// Mitsubishi GX Works2 project: 051023 aula antes de apagar   PLC: Q03UDV

// task Task_01 (event TRUE, interval 0, priority 31): 
// task ST_Example_Safe (event TRUE, interval 0, priority 31): ST_Example_Safe

PROGRAM ST_Example_Safe
VAR
  iDR : INT;
  iHabilitar : BOOL;
  stgOperador : STRING[32];
  iValor01 : INT;
  iValor02 : INT;
END_VAR
iDR:= fEscolherOperacao1( iHabilitar , stgOperador , iValor01 , iValor02 );

iDR:= fEscolherOperacao2( iHabilitar , stgOperador , iValor01 , iValor02 );
END_PROGRAM

FUNCTION fEscolherOperacao1
VAR_INPUT
  xHabilitar : BOOL;
  stgoperador : STRING[32];
  iValor01 : INT;
  iValor02 : INT;
END_VAR
IF xHabilitar THEN 	
	IF  stgoperador="+"  THEN
			 fEscolherOperacao1:=iValor01+iValor02;
	ELSIF stgoperador="-"  THEN
		 fEscolherOperacao1:=iValor01-iValor02;
    ELSIF stgoperador="*"  THEN
		 fEscolherOperacao1:=iValor01*iValor02;
	ELSIF stgoperador="/"  THEN
		 fEscolherOperacao1:=iValor01/iValor02;
	ELSIF (stgoperador="M") OR (stgoperador="M")  THEN
		 fEscolherOperacao1:=iValor01 MOD iValor02;
	ELSE
		fEscolherOperacao1:=32767;
	END_IF;

ELSE
	 fEscolherOperacao1:=-32767;

END_IF;
END_FUNCTION

FUNCTION fEscolherOperacao2
VAR_INPUT
  xHabilitar : BOOL;
  stgoperador : STRING[32];
  iValor01 : INT;
  iValor02 : INT;
END_VAR
CASE  xHabilitar  OF
	 stgoperador="+" :
		 fEscolherOperacao1:=iValor01+iValor02;;
	stgoperador="-" :
		 fEscolherOperacao1:=iValor01-iValor02;
	 stgoperador="*":
		 fEscolherOperacao1:=iValor01*iValor02;
	stgoperador="/":
		fEscolherOperacao1:=iValor01/iValor02;
	(stgoperador="M") OR (stgoperador="M"):
	 fEscolherOperacao1:=iValor01 MOD iValor02;

	ELSE
		fEscolherOperacao1:=32767;
END_CASE;
END_FUNCTION
